TYPE HighLow_pointers :
STRUCT
	pHigh_byte : POINTER TO BYTE;
	pLow_byte : POINTER TO BYTE;
END_STRUCT
END_TYPE

(* stored: Version 1.1.0.1, ProductVersion 3.1.4024.9
   DUT HighLow_pointers: Id {6fe3838e-d0d6-4e5d-a3c6-94a3688164c3} *)
